(* PLC project tni_train, Dassault Systèmes ControlBuild 2024x *)
(* stored: creationDateTime 2023-10-03T11:13:51-01:00 *)

PROGRAM tni_train.tni_train

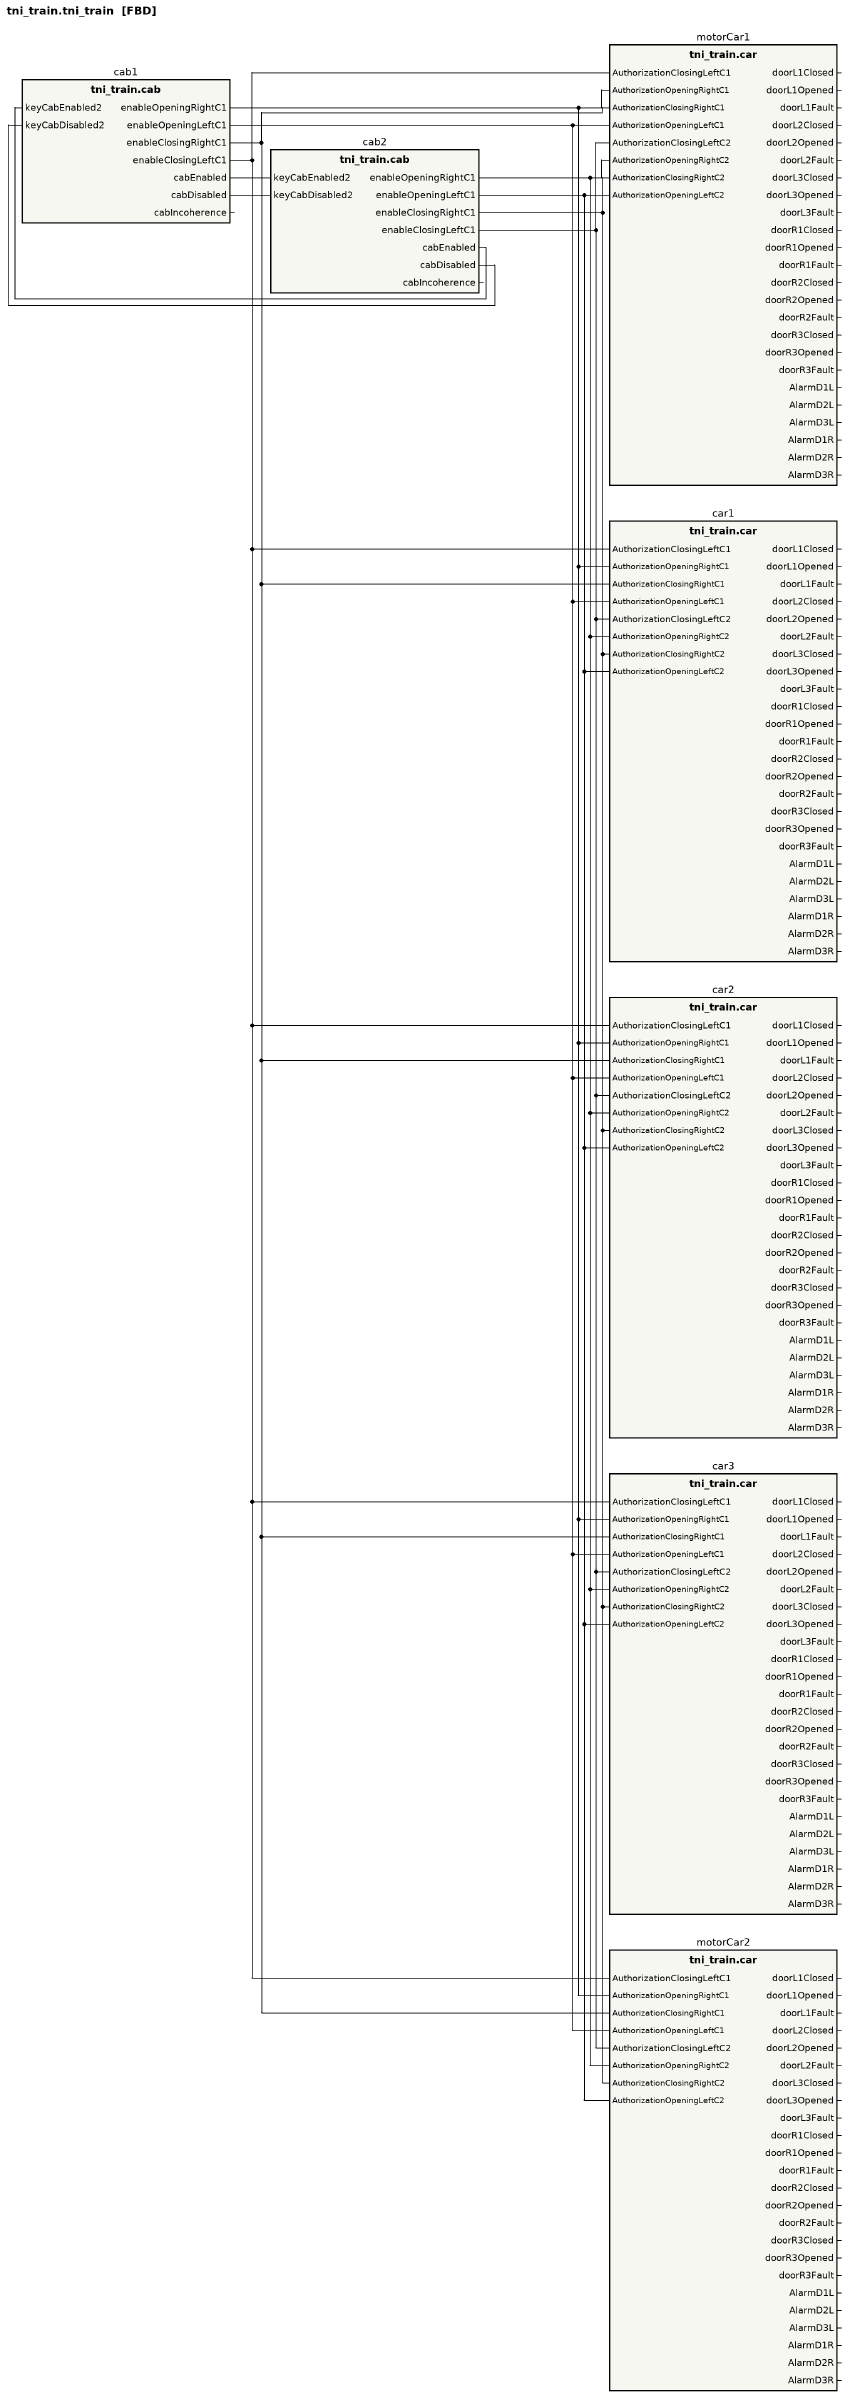
(* FBD diagram, written out as Structured Text *)
cab2(keyCabEnabled2 := cab1.cabEnabled, keyCabDisabled2 := cab1.cabDisabled);
cab1(keyCabEnabled2 := cab2.cabEnabled, keyCabDisabled2 := cab2.cabDisabled);
motorCar1(AuthorizationClosingLeftC1 := cab1.enableClosingLeftC1, AuthorizationOpeningRightC1 := cab1.enableOpeningRightC1, AuthorizationClosingRightC1 := cab1.enableClosingRightC1, AuthorizationOpeningLeftC1 := cab1.enableOpeningLeftC1, AuthorizationClosingLeftC2 := cab2.enableClosingLeftC1, AuthorizationOpeningRightC2 := cab2.enableOpeningRightC1, AuthorizationClosingRightC2 := cab2.enableClosingRightC1, AuthorizationOpeningLeftC2 := cab2.enableOpeningLeftC1);
car1(AuthorizationClosingLeftC1 := cab1.enableClosingLeftC1, AuthorizationOpeningRightC1 := cab1.enableOpeningRightC1, AuthorizationClosingRightC1 := cab1.enableClosingRightC1, AuthorizationOpeningLeftC1 := cab1.enableOpeningLeftC1, AuthorizationClosingLeftC2 := cab2.enableClosingLeftC1, AuthorizationOpeningRightC2 := cab2.enableOpeningRightC1, AuthorizationClosingRightC2 := cab2.enableClosingRightC1, AuthorizationOpeningLeftC2 := cab2.enableOpeningLeftC1);
car2(AuthorizationClosingLeftC1 := cab1.enableClosingLeftC1, AuthorizationOpeningRightC1 := cab1.enableOpeningRightC1, AuthorizationClosingRightC1 := cab1.enableClosingRightC1, AuthorizationOpeningLeftC1 := cab1.enableOpeningLeftC1, AuthorizationClosingLeftC2 := cab2.enableClosingLeftC1, AuthorizationOpeningRightC2 := cab2.enableOpeningRightC1, AuthorizationClosingRightC2 := cab2.enableClosingRightC1, AuthorizationOpeningLeftC2 := cab2.enableOpeningLeftC1);
car3(AuthorizationClosingLeftC1 := cab1.enableClosingLeftC1, AuthorizationOpeningRightC1 := cab1.enableOpeningRightC1, AuthorizationClosingRightC1 := cab1.enableClosingRightC1, AuthorizationOpeningLeftC1 := cab1.enableOpeningLeftC1, AuthorizationClosingLeftC2 := cab2.enableClosingLeftC1, AuthorizationOpeningRightC2 := cab2.enableOpeningRightC1, AuthorizationClosingRightC2 := cab2.enableClosingRightC1, AuthorizationOpeningLeftC2 := cab2.enableOpeningLeftC1);
motorCar2(AuthorizationClosingLeftC1 := cab1.enableClosingLeftC1, AuthorizationOpeningRightC1 := cab1.enableOpeningRightC1, AuthorizationClosingRightC1 := cab1.enableClosingRightC1, AuthorizationOpeningLeftC1 := cab1.enableOpeningLeftC1, AuthorizationClosingLeftC2 := cab2.enableClosingLeftC1, AuthorizationOpeningRightC2 := cab2.enableOpeningRightC1, AuthorizationClosingRightC2 := cab2.enableClosingRightC1, AuthorizationOpeningLeftC2 := cab2.enableOpeningLeftC1);
END_PROGRAM
